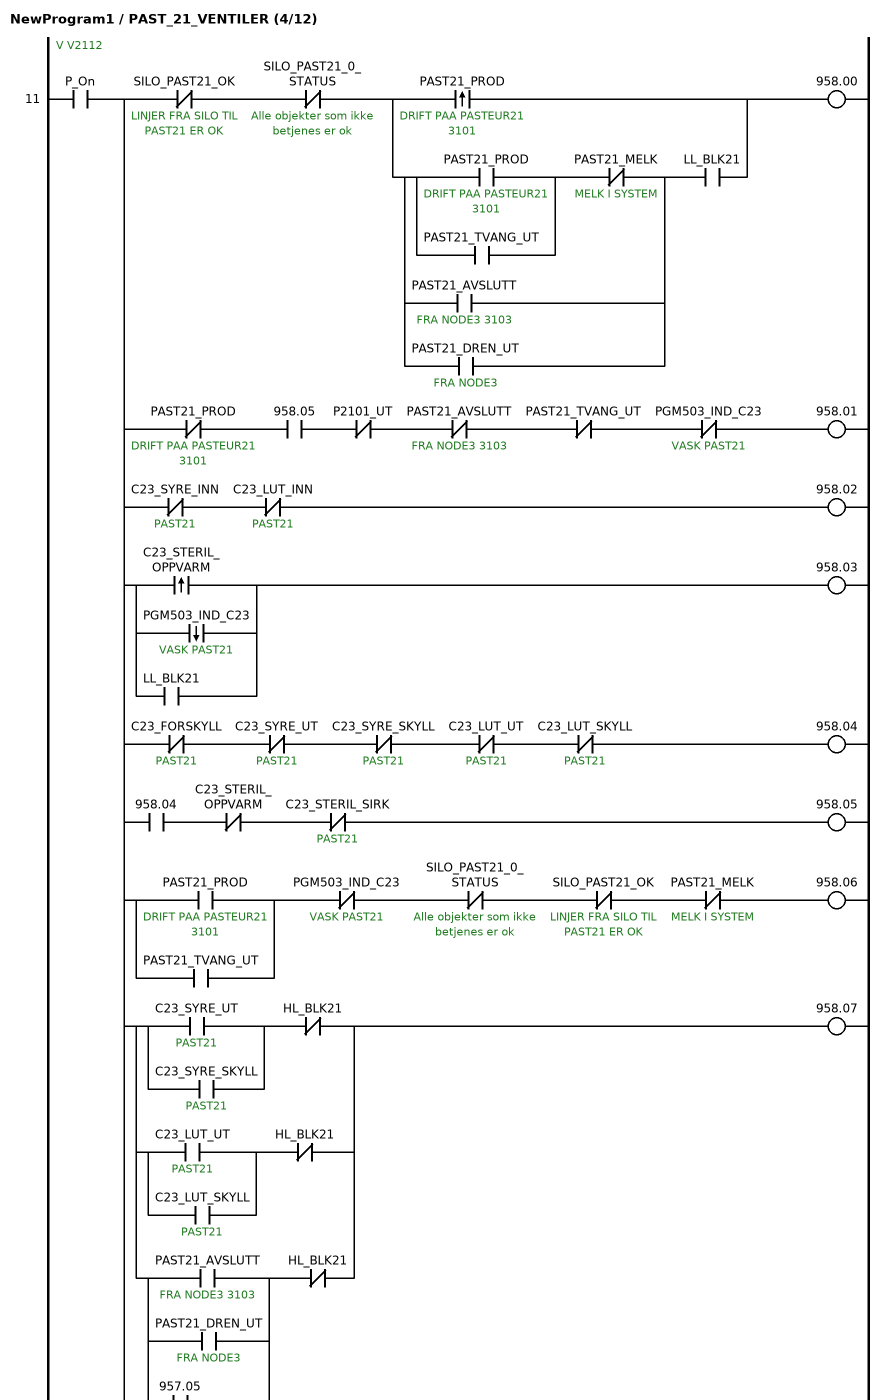
; [picture p1104: NewProgram1 / PAST_21_VENTILER, rungs 11-11]

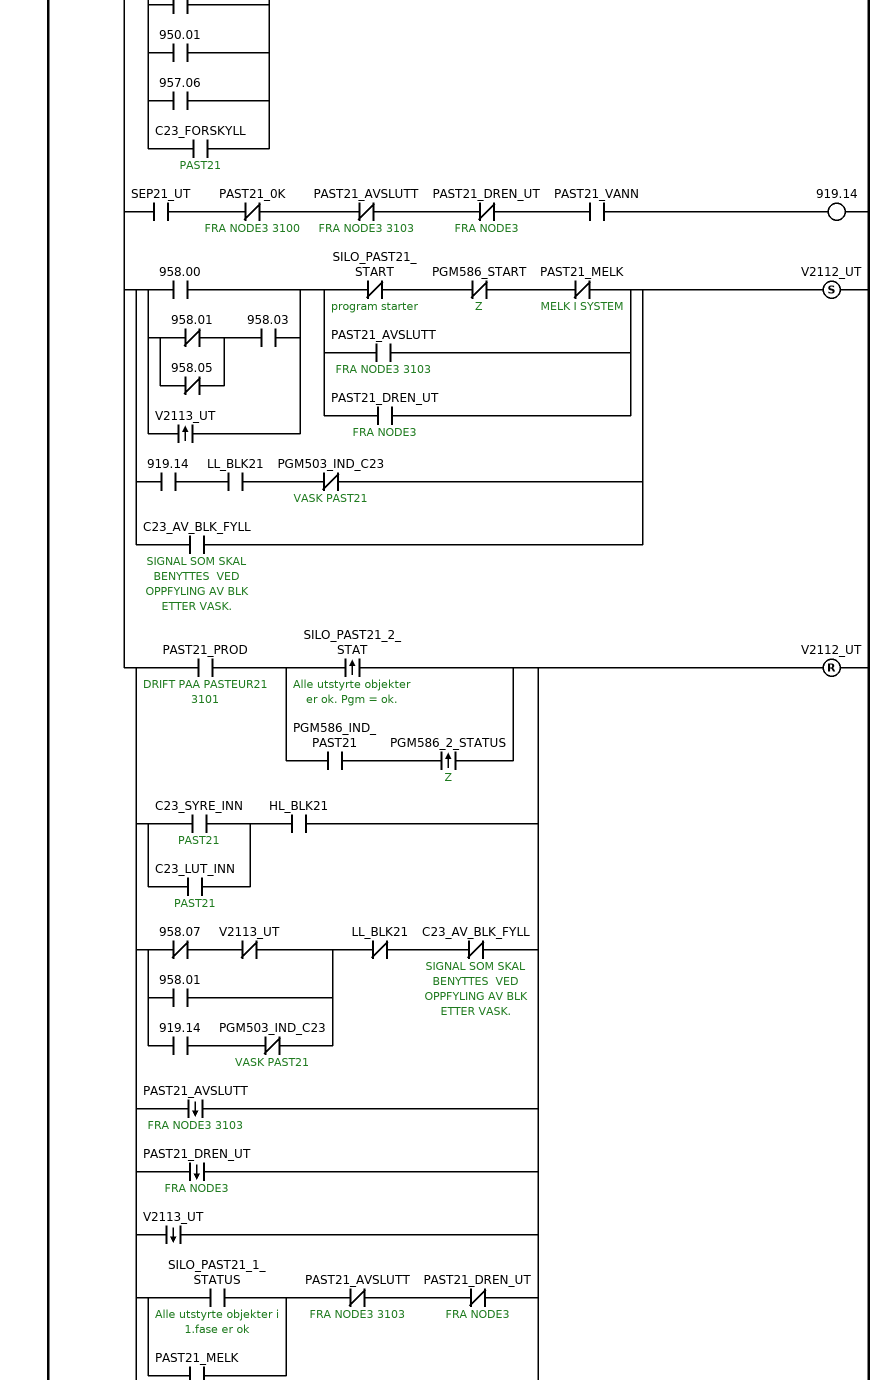

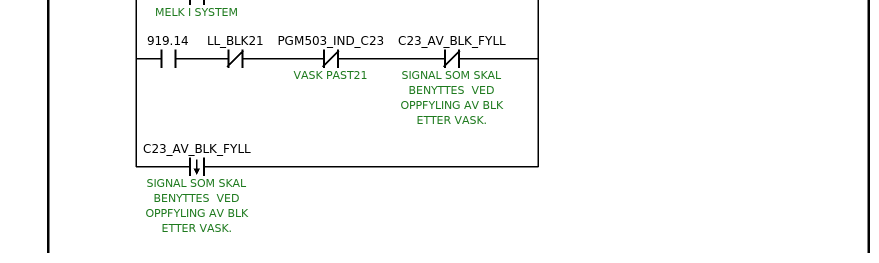
; rung 11: V V2112
LD P_On
OUT TR0
ANDNOT SILO_PAST21_OK  ; LINJER FRA SILO TIL  PAST21 ER OK
ANDNOT SILO_PAST21_0_STATUS  ; Alle objekter som ikke betjenes er ok
@LD PAST21_PROD  ; DRIFT PAA PASTEUR21 3101
LD PAST21_PROD  ; DRIFT PAA PASTEUR21 3101
OR PAST21_TVANG_UT
ANDNOT PAST21_MELK  ; MELK I SYSTEM
OR PAST21_AVSLUTT  ; FRA NODE3 3103
OR PAST21_DREN_UT  ; FRA NODE3
AND LL_BLK21
ORLD
ANDLD
OUT 958.00
LD TR0
ANDNOT PAST21_PROD  ; DRIFT PAA PASTEUR21 3101
AND 958.05
ANDNOT P2101_UT
ANDNOT PAST21_AVSLUTT  ; FRA NODE3 3103
ANDNOT PAST21_TVANG_UT
ANDNOT PGM503_IND_C23  ; VASK PAST21
OUT 958.01
LD TR0
ANDNOT C23_SYRE_INN  ; PAST21
ANDNOT C23_LUT_INN  ; PAST21
OUT 958.02
LD TR0
@LD C23_STERIL_OPPVARM
%OR PGM503_IND_C23  ; VASK PAST21
OR LL_BLK21
ANDLD
OUT 958.03
LD TR0
ANDNOT C23_FORSKYLL  ; PAST21
ANDNOT C23_SYRE_UT  ; PAST21
ANDNOT C23_SYRE_SKYLL  ; PAST21
ANDNOT C23_LUT_UT  ; PAST21
ANDNOT C23_LUT_SKYLL  ; PAST21
OUT 958.04
LD TR0
AND 958.04
ANDNOT C23_STERIL_OPPVARM
ANDNOT C23_STERIL_SIRK  ; PAST21
OUT 958.05
LD TR0
LD PAST21_PROD  ; DRIFT PAA PASTEUR21 3101
OR PAST21_TVANG_UT
ANDLD
ANDNOT PGM503_IND_C23  ; VASK PAST21
ANDNOT SILO_PAST21_0_STATUS  ; Alle objekter som ikke betjenes er ok
ANDNOT SILO_PAST21_OK  ; LINJER FRA SILO TIL  PAST21 ER OK
ANDNOT PAST21_MELK  ; MELK I SYSTEM
OUT 958.06
LD TR0
LD C23_SYRE_UT  ; PAST21
OR C23_SYRE_SKYLL  ; PAST21
ANDNOT HL_BLK21
LD C23_LUT_UT  ; PAST21
OR C23_LUT_SKYLL  ; PAST21
ANDNOT HL_BLK21
ORLD
LD PAST21_AVSLUTT  ; FRA NODE3 3103
OR PAST21_DREN_UT  ; FRA NODE3
OR 957.05
OR 950.01
OR 957.06
OR C23_FORSKYLL  ; PAST21
ANDNOT HL_BLK21
ORLD
ANDLD
OUT 958.07
LD TR0
AND SEP21_UT
ANDNOT PAST21_0K  ; FRA NODE3 3100
ANDNOT PAST21_AVSLUTT  ; FRA NODE3 3103
ANDNOT PAST21_DREN_UT  ; FRA NODE3
AND PAST21_VANN
OUT 919.14
LD TR0
LD 958.00
LDNOT 958.01
ORNOT 958.05
AND 958.03
ORLD
@OR V2113_UT
LDNOT SILO_PAST21_START  ; program starter
ANDNOT PGM586_START  ; Z
ANDNOT PAST21_MELK  ; MELK I SYSTEM
OR PAST21_AVSLUTT  ; FRA NODE3 3103
OR PAST21_DREN_UT  ; FRA NODE3
ANDLD
LD 919.14
AND LL_BLK21
ANDNOT PGM503_IND_C23  ; VASK PAST21
ORLD
OR C23_AV_BLK_FYLL  ; SIGNAL SOM SKAL BENYTTES  VED OPPFYLING AV BLK ETTER VASK.
ANDLD
SET V2112_UT
LD TR0
LD PAST21_PROD  ; DRIFT PAA PASTEUR21 3101
@LD SILO_PAST21_2_STAT  ; Alle utstyrte objekter er ok. Pgm = ok.
LD PGM586_IND_PAST21
@AND PGM586_2_STATUS  ; Z
ORLD
ANDLD
LD C23_SYRE_INN  ; PAST21
OR C23_LUT_INN  ; PAST21
AND HL_BLK21
ORLD
LDNOT 958.07
ANDNOT V2113_UT
OR 958.01
LD 919.14
ANDNOT PGM503_IND_C23  ; VASK PAST21
ORLD
ANDNOT LL_BLK21
ANDNOT C23_AV_BLK_FYLL  ; SIGNAL SOM SKAL BENYTTES  VED OPPFYLING AV BLK ETTER VASK.
ORLD
%OR PAST21_AVSLUTT  ; FRA NODE3 3103
%OR PAST21_DREN_UT  ; FRA NODE3
%OR V2113_UT
LD SILO_PAST21_1_STATUS  ; Alle utstyrte objekter i 1.fase er ok
OR PAST21_MELK  ; MELK I SYSTEM
ANDNOT PAST21_AVSLUTT  ; FRA NODE3 3103
ANDNOT PAST21_DREN_UT  ; FRA NODE3
ORLD
LD 919.14
ANDNOT LL_BLK21
ANDNOT PGM503_IND_C23  ; VASK PAST21
ANDNOT C23_AV_BLK_FYLL  ; SIGNAL SOM SKAL BENYTTES  VED OPPFYLING AV BLK ETTER VASK.
ORLD
%OR C23_AV_BLK_FYLL  ; SIGNAL SOM SKAL BENYTTES  VED OPPFYLING AV BLK ETTER VASK.
ANDLD
RSET V2112_UT

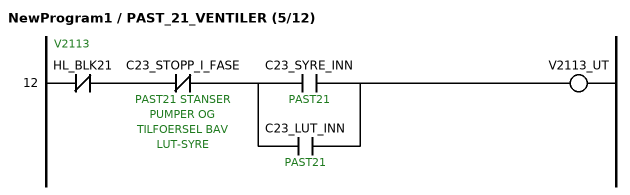
; rung 12: V2113
LDNOT HL_BLK21
ANDNOT C23_STOPP_I_FASE  ; PAST21 STANSER PUMPER OG TILFOERSEL BAV LUT-SYRE
LD C23_SYRE_INN  ; PAST21
OR C23_LUT_INN  ; PAST21
ANDLD
OUT V2113_UT

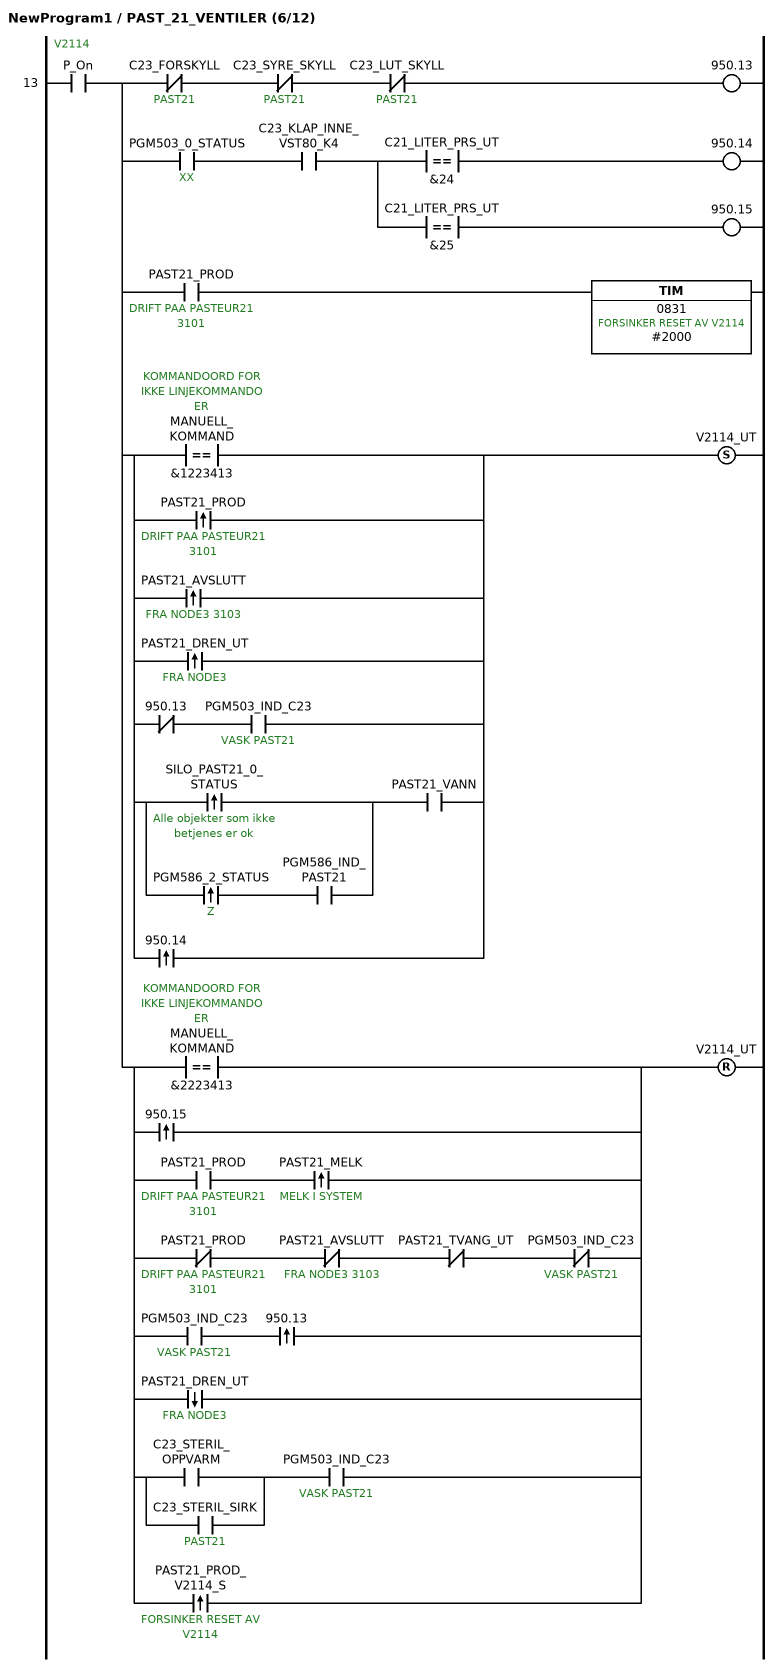
; rung 13: V2114
LD P_On
OUT TR0
ANDNOT C23_FORSKYLL  ; PAST21
ANDNOT C23_SYRE_SKYLL  ; PAST21
ANDNOT C23_LUT_SKYLL  ; PAST21
OUT 950.13
LD TR0
AND PGM503_0_STATUS  ; XX
AND C23_KLAP_INNE_VST80_K4
OUT TR1
AND=(300) C21_LITER_PRS_UT &24
OUT 950.14
LD TR1
AND=(300) C21_LITER_PRS_UT &25
OUT 950.15
LD TR0
AND PAST21_PROD  ; DRIFT PAA PASTEUR21 3101
TIM 0831 #2000  ; FORSINKER RESET AV V2114
LD TR0
LD=L(301) MANUELL_KOMMAND &1223413  ; KOMMANDOORD FOR IKKE LINJEKOMMANDOER
@OR PAST21_PROD  ; DRIFT PAA PASTEUR21 3101
@OR PAST21_AVSLUTT  ; FRA NODE3 3103
@OR PAST21_DREN_UT  ; FRA NODE3
LDNOT 950.13
AND PGM503_IND_C23  ; VASK PAST21
ORLD
@LD SILO_PAST21_0_STATUS  ; Alle objekter som ikke betjenes er ok
@LD PGM586_2_STATUS  ; Z
AND PGM586_IND_PAST21
ORLD
AND PAST21_VANN
ORLD
@OR 950.14
ANDLD
SET V2114_UT
LD TR0
LD=L(301) MANUELL_KOMMAND &2223413  ; KOMMANDOORD FOR IKKE LINJEKOMMANDOER
@OR 950.15
LD PAST21_PROD  ; DRIFT PAA PASTEUR21 3101
@AND PAST21_MELK  ; MELK I SYSTEM
ORLD
LDNOT PAST21_PROD  ; DRIFT PAA PASTEUR21 3101
ANDNOT PAST21_AVSLUTT  ; FRA NODE3 3103
ANDNOT PAST21_TVANG_UT
ANDNOT PGM503_IND_C23  ; VASK PAST21
ORLD
LD PGM503_IND_C23  ; VASK PAST21
@AND 950.13
ORLD
%OR PAST21_DREN_UT  ; FRA NODE3
LD C23_STERIL_OPPVARM
OR C23_STERIL_SIRK  ; PAST21
AND PGM503_IND_C23  ; VASK PAST21
ORLD
@OR PAST21_PROD_V2114_S  ; FORSINKER RESET AV V2114
ANDLD
RSET V2114_UT

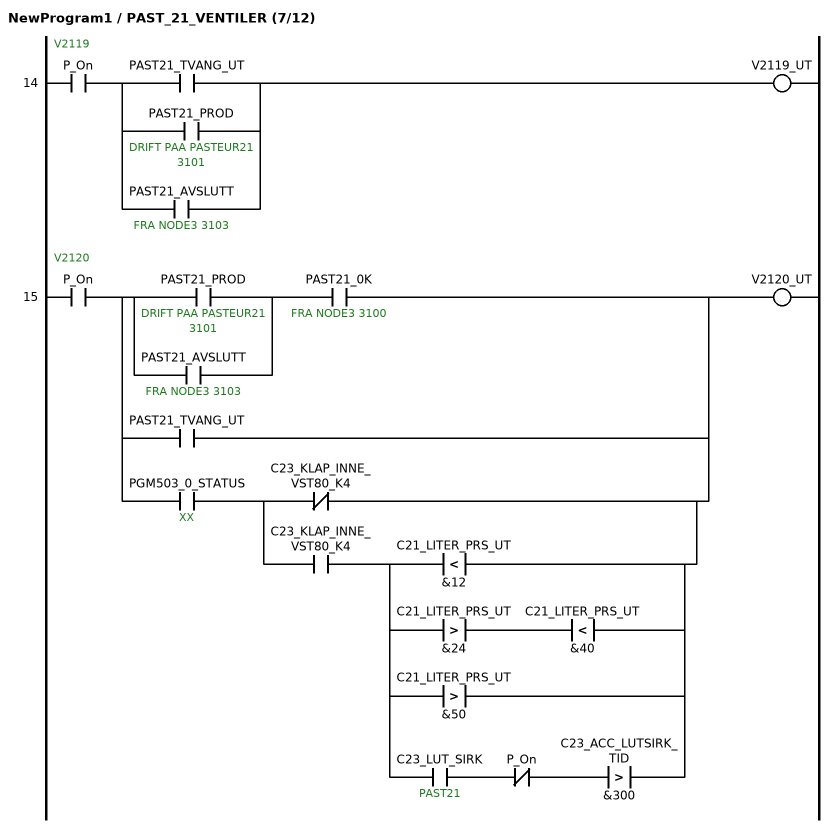
; rung 14: V2119
LD P_On
LD PAST21_TVANG_UT
OR PAST21_PROD  ; DRIFT PAA PASTEUR21 3101
OR PAST21_AVSLUTT  ; FRA NODE3 3103
ANDLD
OUT V2119_UT
; rung 15: V2120
LD P_On
LD PAST21_PROD  ; DRIFT PAA PASTEUR21 3101
OR PAST21_AVSLUTT  ; FRA NODE3 3103
AND PAST21_0K  ; FRA NODE3 3100
OR PAST21_TVANG_UT
LD PGM503_0_STATUS  ; XX
LDNOT C23_KLAP_INNE_VST80_K4
LD C23_KLAP_INNE_VST80_K4
LD<(310) C21_LITER_PRS_UT &12
LD>(320) C21_LITER_PRS_UT &24
AND<(310) C21_LITER_PRS_UT &40
ORLD
OR>(320) C21_LITER_PRS_UT &50
LD C23_LUT_SIRK  ; PAST21
ANDNOT P_On
AND>(320) C23_ACC_LUTSIRK_TID &300
ORLD
ANDLD
ORLD
ANDLD
ORLD
ANDLD
OUT V2120_UT

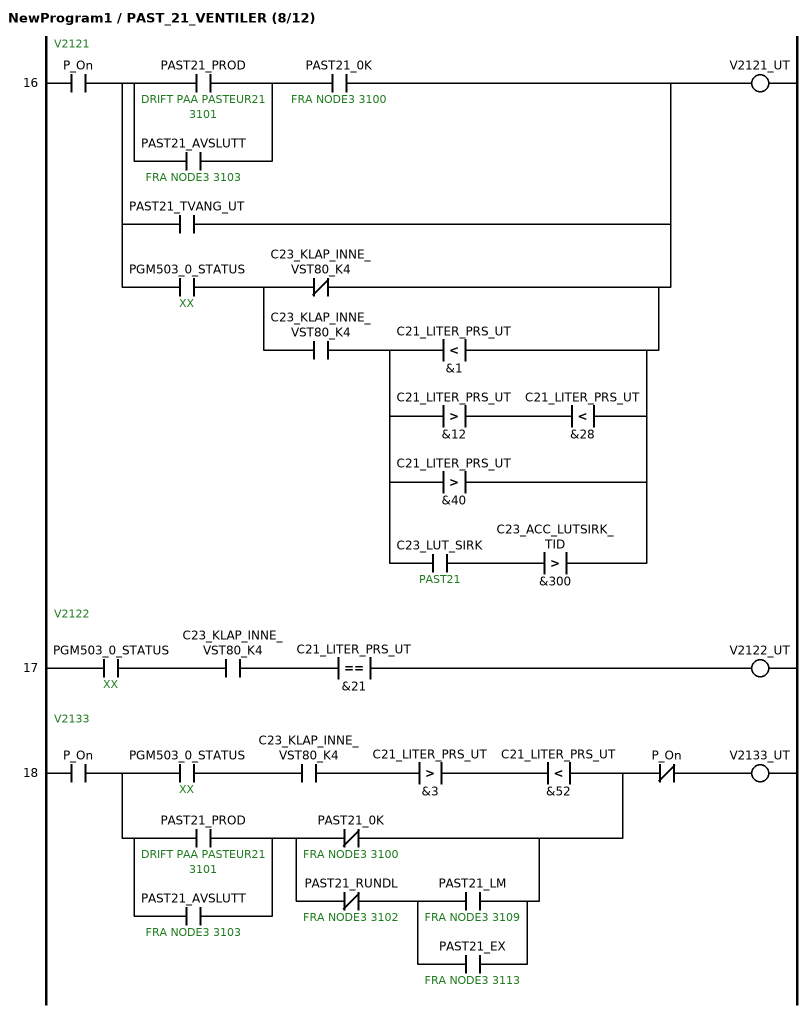
; rung 16: V2121
LD P_On
LD PAST21_PROD  ; DRIFT PAA PASTEUR21 3101
OR PAST21_AVSLUTT  ; FRA NODE3 3103
AND PAST21_0K  ; FRA NODE3 3100
OR PAST21_TVANG_UT
LD PGM503_0_STATUS  ; XX
LDNOT C23_KLAP_INNE_VST80_K4
LD C23_KLAP_INNE_VST80_K4
LD<(310) C21_LITER_PRS_UT &1
LD>(320) C21_LITER_PRS_UT &12
AND<(310) C21_LITER_PRS_UT &28
ORLD
OR>(320) C21_LITER_PRS_UT &40
LD C23_LUT_SIRK  ; PAST21
AND>(320) C23_ACC_LUTSIRK_TID &300
ORLD
ANDLD
ORLD
ANDLD
ORLD
ANDLD
OUT V2121_UT
; rung 17: V2122
LD PGM503_0_STATUS  ; XX
AND C23_KLAP_INNE_VST80_K4
AND=(300) C21_LITER_PRS_UT &21
OUT V2122_UT
; rung 18: V2133
LD P_On
LD PGM503_0_STATUS  ; XX
AND C23_KLAP_INNE_VST80_K4
AND>(320) C21_LITER_PRS_UT &3
AND<(310) C21_LITER_PRS_UT &52
LD PAST21_PROD  ; DRIFT PAA PASTEUR21 3101
OR PAST21_AVSLUTT  ; FRA NODE3 3103
LDNOT PAST21_0K  ; FRA NODE3 3100
LDNOT PAST21_RUNDL  ; FRA NODE3 3102
LD PAST21_LM  ; FRA NODE3 3109
OR PAST21_EX  ; FRA NODE3 3113
ANDLD
ORLD
ANDLD
ORLD
ANDLD
ANDNOT P_On
OUT V2133_UT

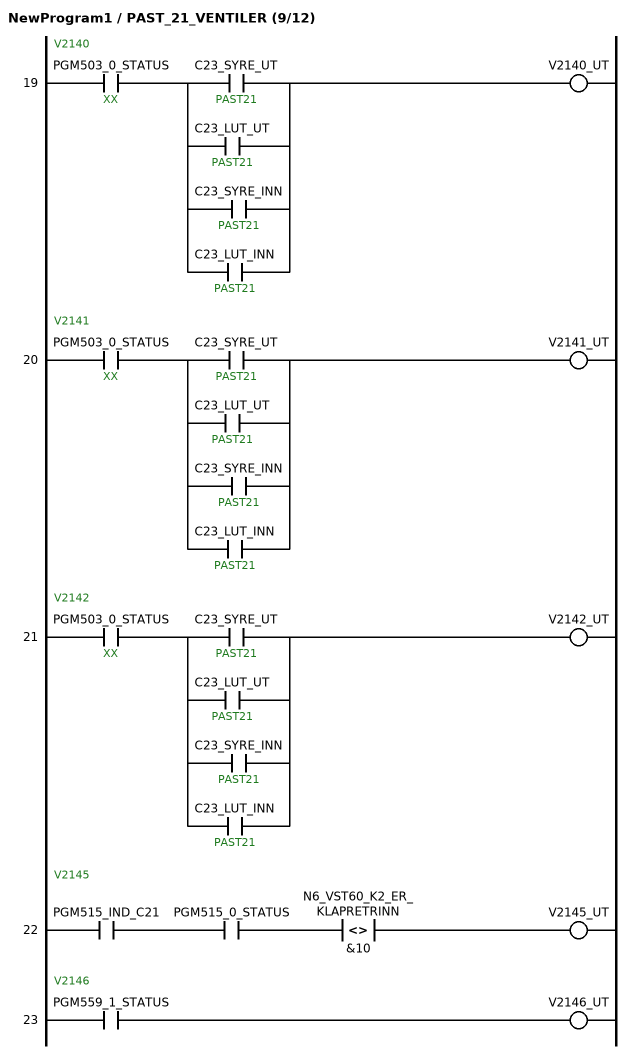
; rung 19: V2140
LD PGM503_0_STATUS  ; XX
LD C23_SYRE_UT  ; PAST21
OR C23_LUT_UT  ; PAST21
OR C23_SYRE_INN  ; PAST21
OR C23_LUT_INN  ; PAST21
ANDLD
OUT V2140_UT
; rung 20: V2141
LD PGM503_0_STATUS  ; XX
LD C23_SYRE_UT  ; PAST21
OR C23_LUT_UT  ; PAST21
OR C23_SYRE_INN  ; PAST21
OR C23_LUT_INN  ; PAST21
ANDLD
OUT V2141_UT
; rung 21: V2142
LD PGM503_0_STATUS  ; XX
LD C23_SYRE_UT  ; PAST21
OR C23_LUT_UT  ; PAST21
OR C23_SYRE_INN  ; PAST21
OR C23_LUT_INN  ; PAST21
ANDLD
OUT V2142_UT
; rung 22: V2145
LD PGM515_IND_C21
AND PGM515_0_STATUS
AND<>(305) N6_VST60_K2_ER_KLAPRETRINN &10
OUT V2145_UT
; rung 23: V2146
LD PGM559_1_STATUS
OUT V2146_UT

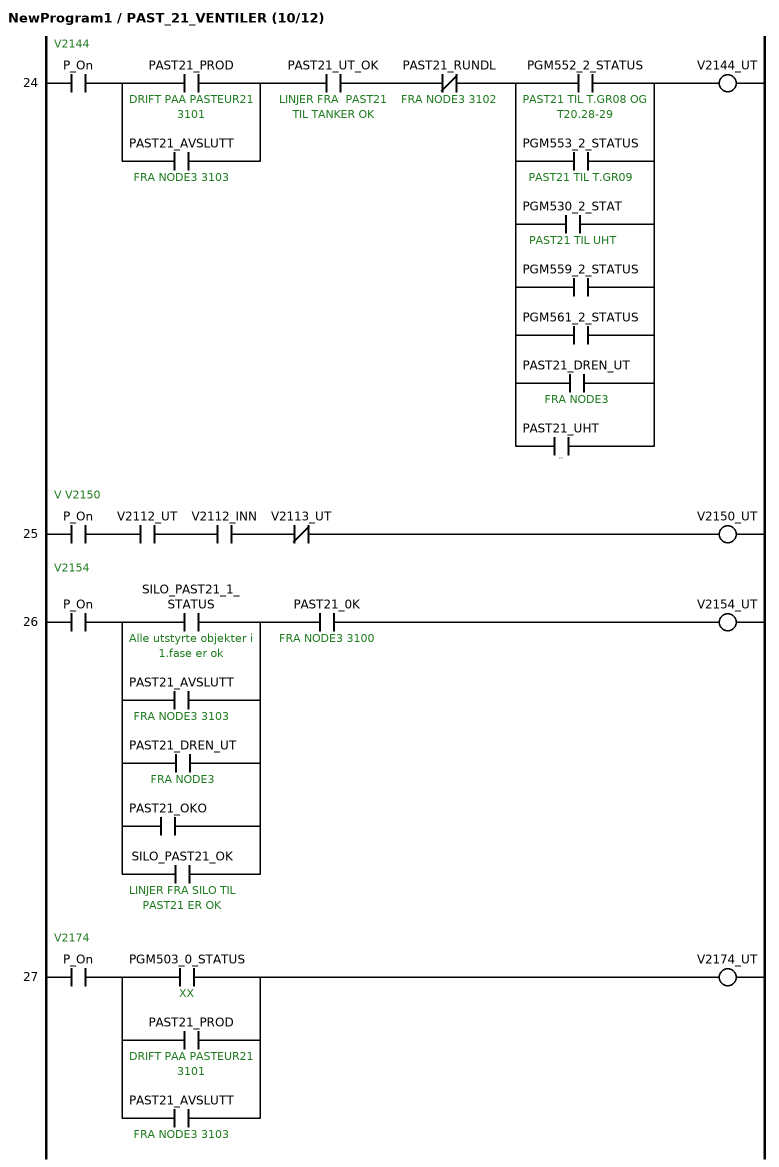
; rung 24: V2144
LD P_On
LD PAST21_PROD  ; DRIFT PAA PASTEUR21 3101
OR PAST21_AVSLUTT  ; FRA NODE3 3103
ANDLD
AND PAST21_UT_OK  ; LINJER FRA  PAST21 TIL TANKER OK
ANDNOT PAST21_RUNDL  ; FRA NODE3 3102
LD PGM552_2_STATUS  ; PAST21 TIL T.GR08 OG T20.28-29
OR PGM553_2_STATUS  ; PAST21 TIL T.GR09
OR PGM530_2_STAT  ; PAST21 TIL UHT
OR PGM559_2_STATUS
OR PGM561_2_STATUS
OR PAST21_DREN_UT  ; FRA NODE3
OR PAST21_UHT  ; ¨
ANDLD
OUT V2144_UT
; rung 25: V V2150
LD P_On
AND V2112_UT
AND V2112_INN
ANDNOT V2113_UT
OUT V2150_UT
; rung 26: V2154
LD P_On
LD SILO_PAST21_1_STATUS  ; Alle utstyrte objekter i 1.fase er ok
OR PAST21_AVSLUTT  ; FRA NODE3 3103
OR PAST21_DREN_UT  ; FRA NODE3
OR PAST21_OKO
OR SILO_PAST21_OK  ; LINJER FRA SILO TIL  PAST21 ER OK
ANDLD
AND PAST21_0K  ; FRA NODE3 3100
OUT V2154_UT
; rung 27: V2174
LD P_On
LD PGM503_0_STATUS  ; XX
OR PAST21_PROD  ; DRIFT PAA PASTEUR21 3101
OR PAST21_AVSLUTT  ; FRA NODE3 3103
ANDLD
OUT V2174_UT

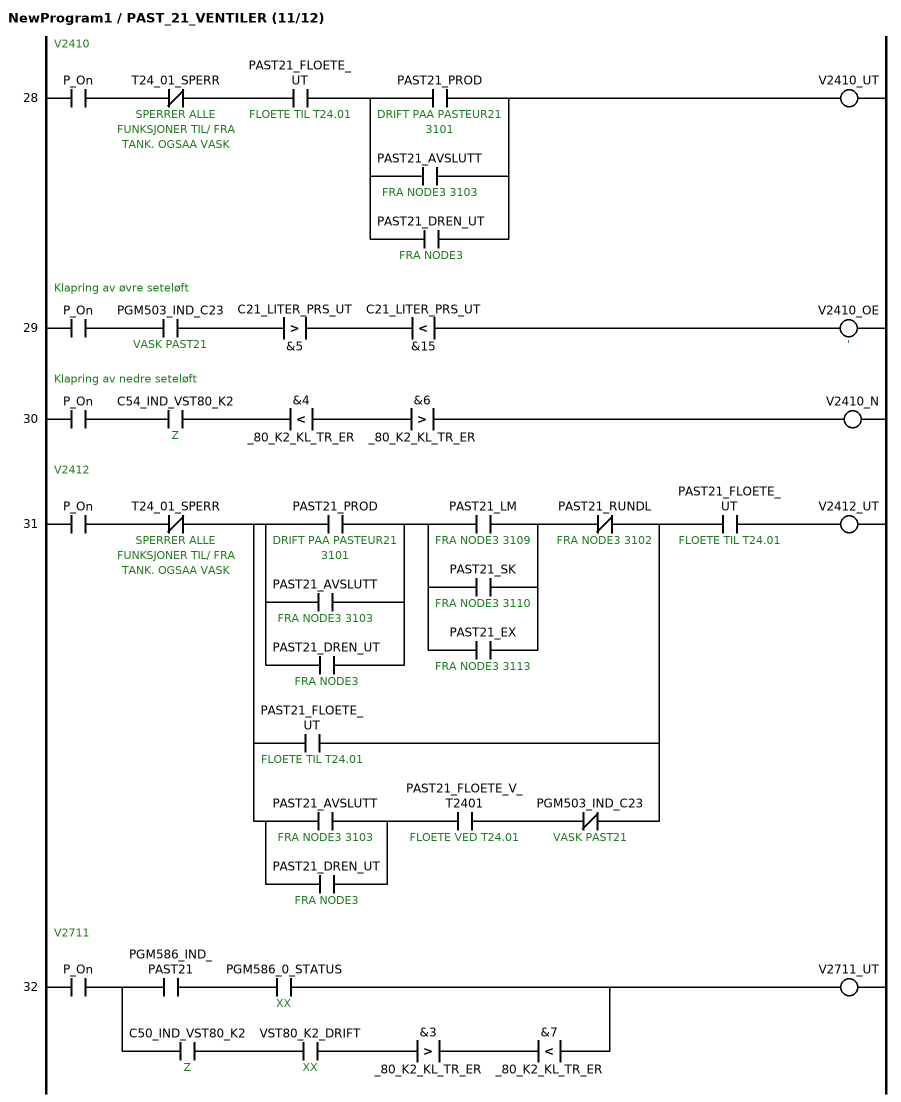
; rung 28: V2410
LD P_On
ANDNOT T24_01_SPERR  ; SPERRER ALLE FUNKSJONER TIL/ FRA TANK. OGSAA VASK
AND PAST21_FLOETE_UT  ; FLOETE TIL T24.01
LD PAST21_PROD  ; DRIFT PAA PASTEUR21 3101
OR PAST21_AVSLUTT  ; FRA NODE3 3103
OR PAST21_DREN_UT  ; FRA NODE3
ANDLD
OUT V2410_UT
; rung 29: Klapring av øvre seteløft
LD P_On
AND PGM503_IND_C23  ; VASK PAST21
AND>(320) C21_LITER_PRS_UT &5
AND<(310) C21_LITER_PRS_UT &15
OUT V2410_OE  ; '
; rung 30: Klapring av nedre seteløft
LD P_On
AND C54_IND_VST80_K2  ; Z
AND<(310) &4 _80_K2_KL_TR_ER
AND>(320) &6 _80_K2_KL_TR_ER
OUT V2410_N
; rung 31: V2412
LD P_On
ANDNOT T24_01_SPERR  ; SPERRER ALLE FUNKSJONER TIL/ FRA TANK. OGSAA VASK
LD PAST21_PROD  ; DRIFT PAA PASTEUR21 3101
OR PAST21_AVSLUTT  ; FRA NODE3 3103
OR PAST21_DREN_UT  ; FRA NODE3
LD PAST21_LM  ; FRA NODE3 3109
OR PAST21_SK  ; FRA NODE3 3110
OR PAST21_EX  ; FRA NODE3 3113
ANDLD
ANDNOT PAST21_RUNDL  ; FRA NODE3 3102
OR PAST21_FLOETE_UT  ; FLOETE TIL T24.01
LD PAST21_AVSLUTT  ; FRA NODE3 3103
OR PAST21_DREN_UT  ; FRA NODE3
AND PAST21_FLOETE_V_T2401  ; FLOETE VED T24.01
ANDNOT PGM503_IND_C23  ; VASK PAST21
ORLD
ANDLD
AND PAST21_FLOETE_UT  ; FLOETE TIL T24.01
OUT V2412_UT
; rung 32: V2711
LD P_On
LD PGM586_IND_PAST21
AND PGM586_0_STATUS  ; XX
LD C50_IND_VST80_K2  ; Z
AND VST80_K2_DRIFT  ; XX
AND>(320) &3 _80_K2_KL_TR_ER
AND<(310) &7 _80_K2_KL_TR_ER
ORLD
ANDLD
OUT V2711_UT

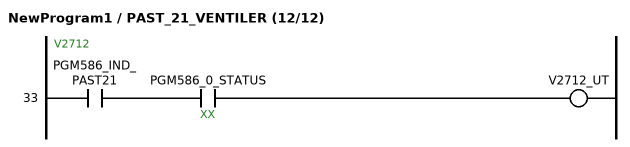
; rung 33: V2712
LD PGM586_IND_PAST21
AND PGM586_0_STATUS  ; XX
OUT V2712_UT

### Section PAST_21_SKRIVER

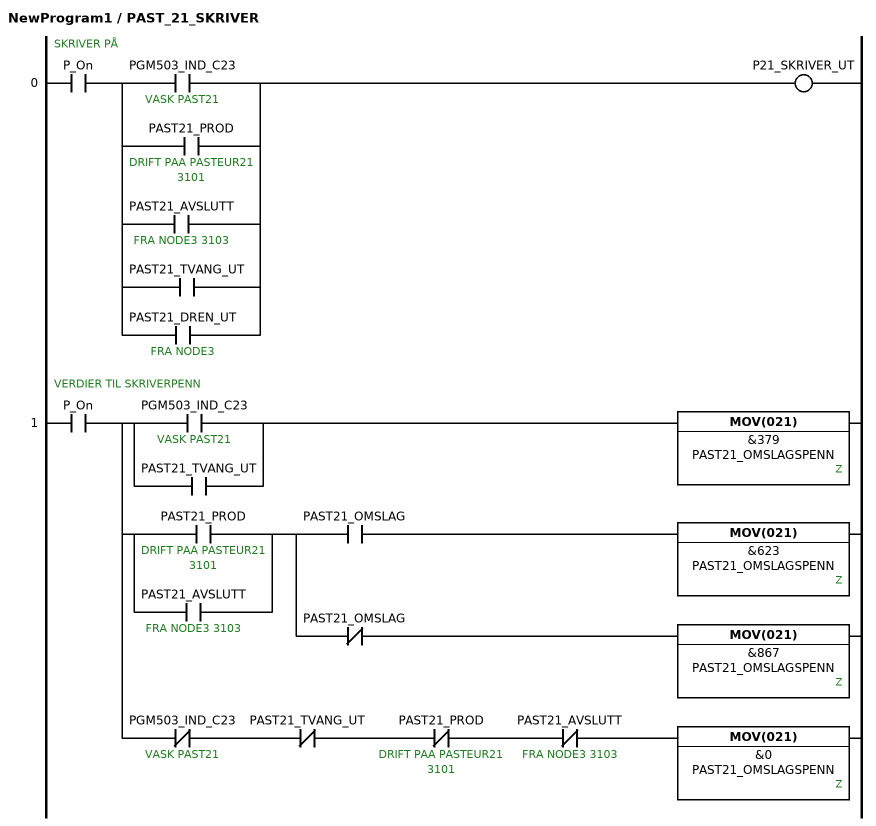
; rung 0: SKRIVER PÅ
LD P_On
LD PGM503_IND_C23  ; VASK PAST21
OR PAST21_PROD  ; DRIFT PAA PASTEUR21 3101
OR PAST21_AVSLUTT  ; FRA NODE3 3103
OR PAST21_TVANG_UT
OR PAST21_DREN_UT  ; FRA NODE3
ANDLD
OUT P21_SKRIVER_UT
; rung 1: VERDIER TIL SKRIVERPENN
LD P_On
OUT TR0
LD PGM503_IND_C23  ; VASK PAST21
OR PAST21_TVANG_UT
ANDLD
MOV(021) &379 PAST21_OMSLAGSPENN  ; Z
LD TR0
LD PAST21_PROD  ; DRIFT PAA PASTEUR21 3101
OR PAST21_AVSLUTT  ; FRA NODE3 3103
ANDLD
OUT TR1
AND PAST21_OMSLAG
MOV(021) &623 PAST21_OMSLAGSPENN  ; Z
LD TR1
ANDNOT PAST21_OMSLAG
MOV(021) &867 PAST21_OMSLAGSPENN  ; Z
LD TR0
ANDNOT PGM503_IND_C23  ; VASK PAST21
ANDNOT PAST21_TVANG_UT
ANDNOT PAST21_PROD  ; DRIFT PAA PASTEUR21 3101
ANDNOT PAST21_AVSLUTT  ; FRA NODE3 3103
MOV(021) &0 PAST21_OMSLAGSPENN  ; Z

### Section PAST_21_TELLERFUNKSJONER

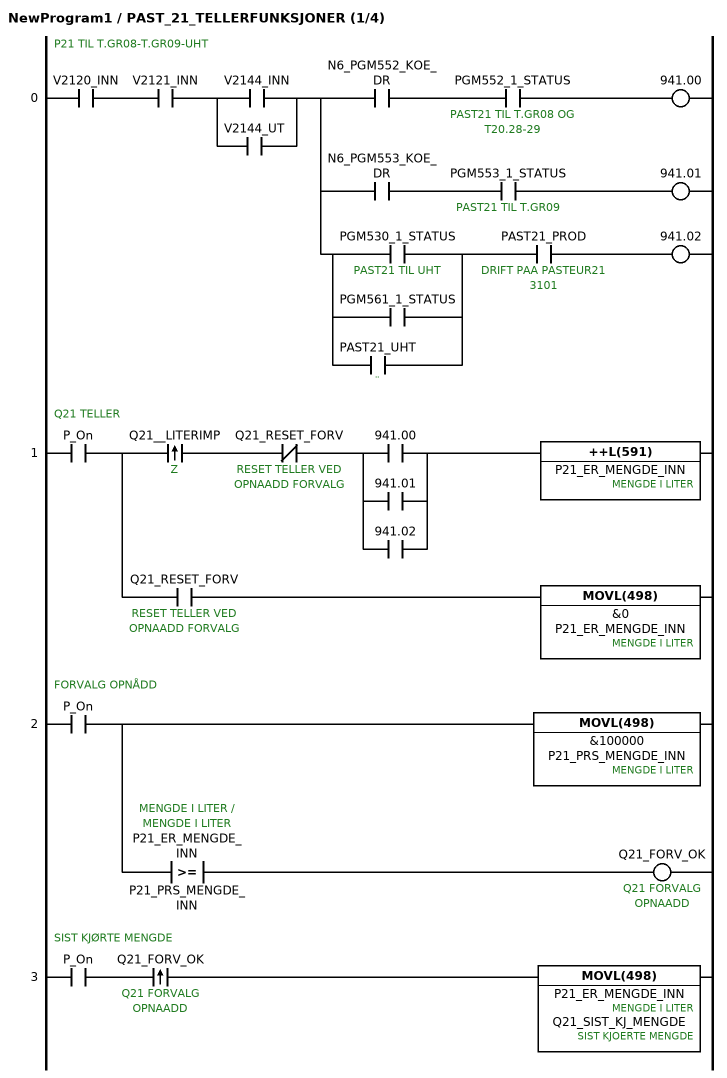
; rung 0: P21 TIL T.GR08-T.GR09-UHT
LD V2120_INN
AND V2121_INN
LD V2144_INN
OR V2144_UT
ANDLD
OUT TR0
AND N6_PGM552_KOE_DR
AND PGM552_1_STATUS  ; PAST21 TIL T.GR08 OG T20.28-29
OUT 941.00
LD TR0
AND N6_PGM553_KOE_DR
AND PGM553_1_STATUS  ; PAST21 TIL T.GR09
OUT 941.01
LD TR0
LD PGM530_1_STATUS  ; PAST21 TIL UHT
OR PGM561_1_STATUS
OR PAST21_UHT  ; ¨
ANDLD
AND PAST21_PROD  ; DRIFT PAA PASTEUR21 3101
OUT 941.02
; rung 1: Q21 TELLER
LD P_On
OUT TR0
@AND Q21__LITERIMP  ; Z
ANDNOT Q21_RESET_FORV  ; RESET TELLER VED OPNAADD FORVALG
LD 941.00
OR 941.01
OR 941.02
ANDLD
++L(591) P21_ER_MENGDE_INN  ; MENGDE I LITER
LD TR0
AND Q21_RESET_FORV  ; RESET TELLER VED OPNAADD FORVALG
MOVL(498) &0 P21_ER_MENGDE_INN  ; MENGDE I LITER
; rung 2: FORVALG OPNÅDD
LD P_On
MOVL(498) &100000 P21_PRS_MENGDE_INN  ; MENGDE I LITER
AND>=L(326) P21_ER_MENGDE_INN P21_PRS_MENGDE_INN  ; MENGDE I LITER
OUT Q21_FORV_OK  ; Q21 FORVALG OPNAADD
; rung 3: SIST KJØRTE MENGDE
LD P_On
@AND Q21_FORV_OK  ; Q21 FORVALG OPNAADD
MOVL(498) P21_ER_MENGDE_INN Q21_SIST_KJ_MENGDE  ; MENGDE I LITER, SIST KJOERTE MENGDE

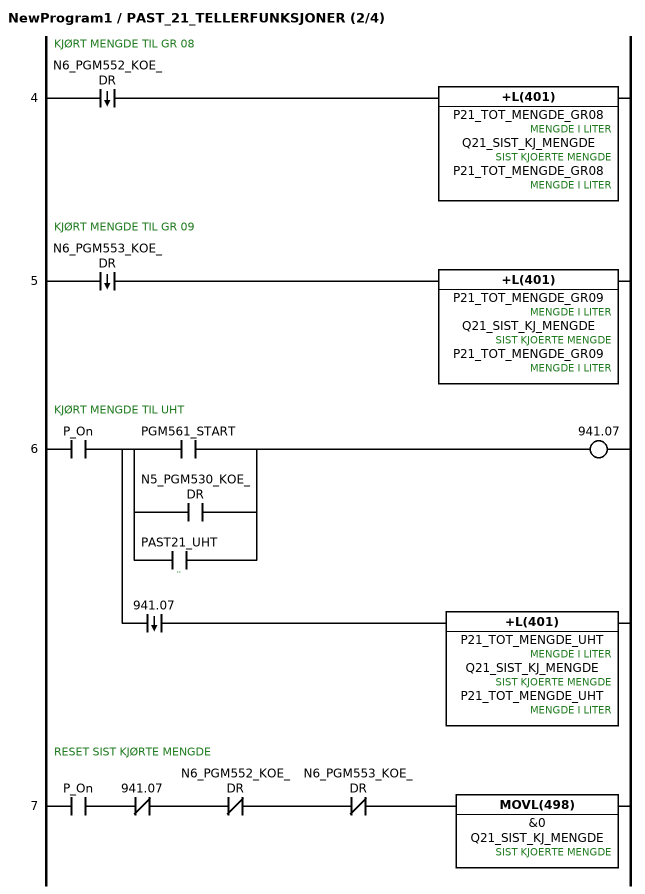
; rung 4: KJØRT MENGDE TIL GR 08
%LD N6_PGM552_KOE_DR
+L(401) P21_TOT_MENGDE_GR08 Q21_SIST_KJ_MENGDE P21_TOT_MENGDE_GR08  ; MENGDE I LITER, SIST KJOERTE MENGDE
; rung 5: KJØRT MENGDE TIL GR 09
%LD N6_PGM553_KOE_DR
+L(401) P21_TOT_MENGDE_GR09 Q21_SIST_KJ_MENGDE P21_TOT_MENGDE_GR09  ; MENGDE I LITER, SIST KJOERTE MENGDE
; rung 6: KJØRT MENGDE TIL UHT
LD P_On
OUT TR0
LD PGM561_START
OR N5_PGM530_KOE_DR
OR PAST21_UHT  ; ¨
ANDLD
OUT 941.07
LD TR0
%AND 941.07
+L(401) P21_TOT_MENGDE_UHT Q21_SIST_KJ_MENGDE P21_TOT_MENGDE_UHT  ; MENGDE I LITER, SIST KJOERTE MENGDE
; rung 7: RESET SIST KJØRTE MENGDE
LD P_On
ANDNOT 941.07
ANDNOT N6_PGM552_KOE_DR
ANDNOT N6_PGM553_KOE_DR
MOVL(498) &0 Q21_SIST_KJ_MENGDE  ; SIST KJOERTE MENGDE

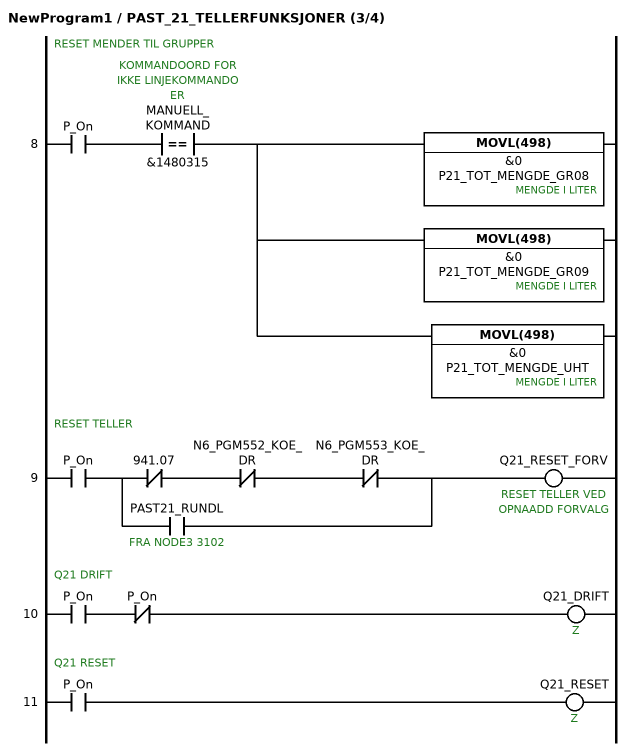
; rung 8: RESET MENDER TIL GRUPPER
LD P_On
AND=L(301) MANUELL_KOMMAND &1480315  ; KOMMANDOORD FOR IKKE LINJEKOMMANDOER
MOVL(498) &0 P21_TOT_MENGDE_GR08  ; MENGDE I LITER
MOVL(498) &0 P21_TOT_MENGDE_GR09  ; MENGDE I LITER
MOVL(498) &0 P21_TOT_MENGDE_UHT  ; MENGDE I LITER
; rung 9: RESET TELLER
LD P_On
LDNOT 941.07
ANDNOT N6_PGM552_KOE_DR
ANDNOT N6_PGM553_KOE_DR
OR PAST21_RUNDL  ; FRA NODE3 3102
ANDLD
OUT Q21_RESET_FORV  ; RESET TELLER VED OPNAADD FORVALG
; rung 10: Q21 DRIFT
LD P_On
ANDNOT P_On
OUT Q21_DRIFT  ; Z
; rung 11: Q21 RESET
LD P_On
OUT Q21_RESET  ; Z

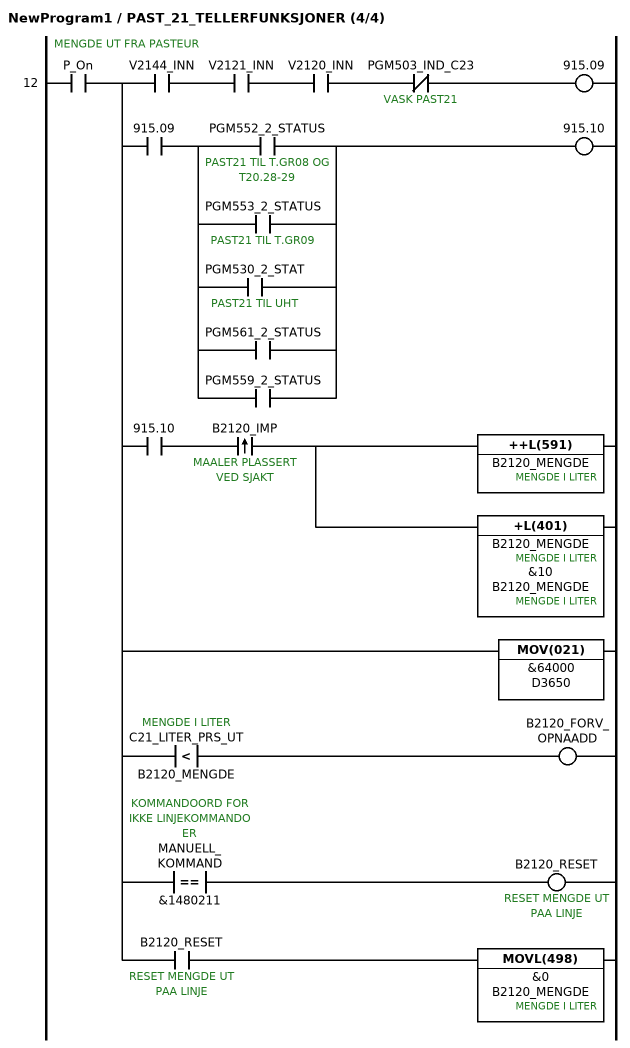
; rung 12: MENGDE UT FRA PASTEUR
LD P_On
OUT TR0
AND V2144_INN
AND V2121_INN
AND V2120_INN
ANDNOT PGM503_IND_C23  ; VASK PAST21
OUT 915.09
LD TR0
AND 915.09
LD PGM552_2_STATUS  ; PAST21 TIL T.GR08 OG T20.28-29
OR PGM553_2_STATUS  ; PAST21 TIL T.GR09
OR PGM530_2_STAT  ; PAST21 TIL UHT
OR PGM561_2_STATUS
OR PGM559_2_STATUS
ANDLD
OUT 915.10
LD TR0
AND 915.10
@AND B2120_IMP  ; MAALER PLASSERT VED SJAKT
++L(591) B2120_MENGDE  ; MENGDE I LITER
+L(401) B2120_MENGDE &10 B2120_MENGDE  ; MENGDE I LITER
LD TR0
MOV(021) &64000 D3650
AND<L(311) C21_LITER_PRS_UT B2120_MENGDE  ; MENGDE I LITER
OUT B2120_FORV_OPNAADD
LD TR0
AND=L(301) MANUELL_KOMMAND &1480211  ; KOMMANDOORD FOR IKKE LINJEKOMMANDOER
OUT B2120_RESET  ; RESET MENGDE UT PAA LINJE
LD TR0
AND B2120_RESET  ; RESET MENGDE UT PAA LINJE
MOVL(498) &0 B2120_MENGDE  ; MENGDE I LITER

### Section P21_MELK_IRØR_TIL_TGR

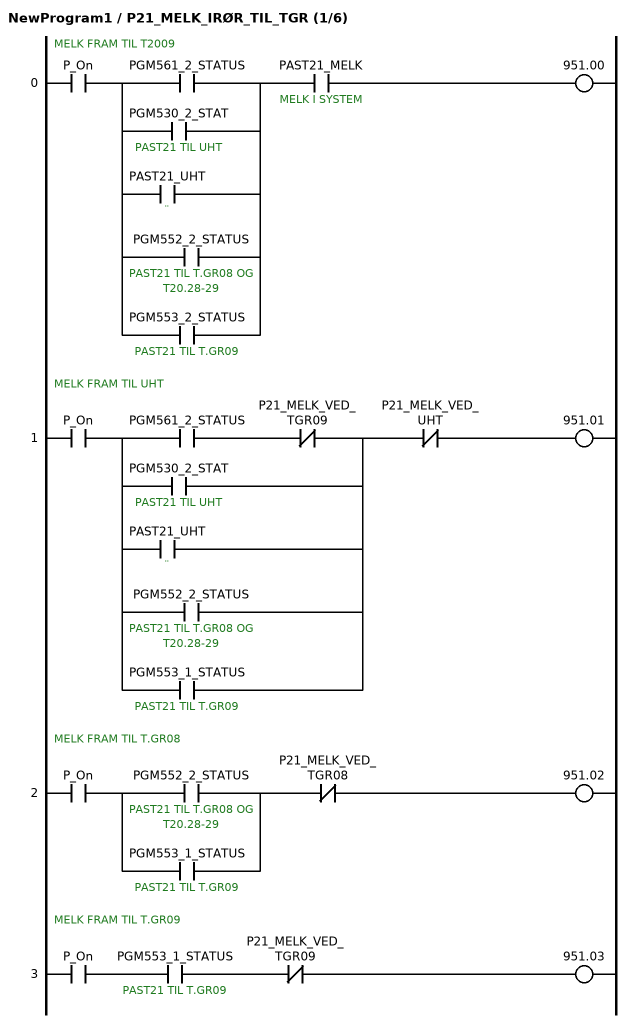
; rung 0: MELK FRAM TIL T2009
LD P_On
LD PGM561_2_STATUS
OR PGM530_2_STAT  ; PAST21 TIL UHT
OR PAST21_UHT  ; ¨
OR PGM552_2_STATUS  ; PAST21 TIL T.GR08 OG T20.28-29
OR PGM553_2_STATUS  ; PAST21 TIL T.GR09
ANDLD
AND PAST21_MELK  ; MELK I SYSTEM
OUT 951.00
; rung 1: MELK FRAM TIL UHT
LD P_On
LD PGM561_2_STATUS
ANDNOT P21_MELK_VED_TGR09
OR PGM530_2_STAT  ; PAST21 TIL UHT
OR PAST21_UHT  ; ¨
OR PGM552_2_STATUS  ; PAST21 TIL T.GR08 OG T20.28-29
OR PGM553_1_STATUS  ; PAST21 TIL T.GR09
ANDLD
ANDNOT P21_MELK_VED_UHT
OUT 951.01
; rung 2: MELK FRAM TIL T.GR08
LD P_On
LD PGM552_2_STATUS  ; PAST21 TIL T.GR08 OG T20.28-29
OR PGM553_1_STATUS  ; PAST21 TIL T.GR09
ANDLD
ANDNOT P21_MELK_VED_TGR08
OUT 951.02
; rung 3: MELK FRAM TIL T.GR09
LD P_On
AND PGM553_1_STATUS  ; PAST21 TIL T.GR09
ANDNOT P21_MELK_VED_TGR09
OUT 951.03

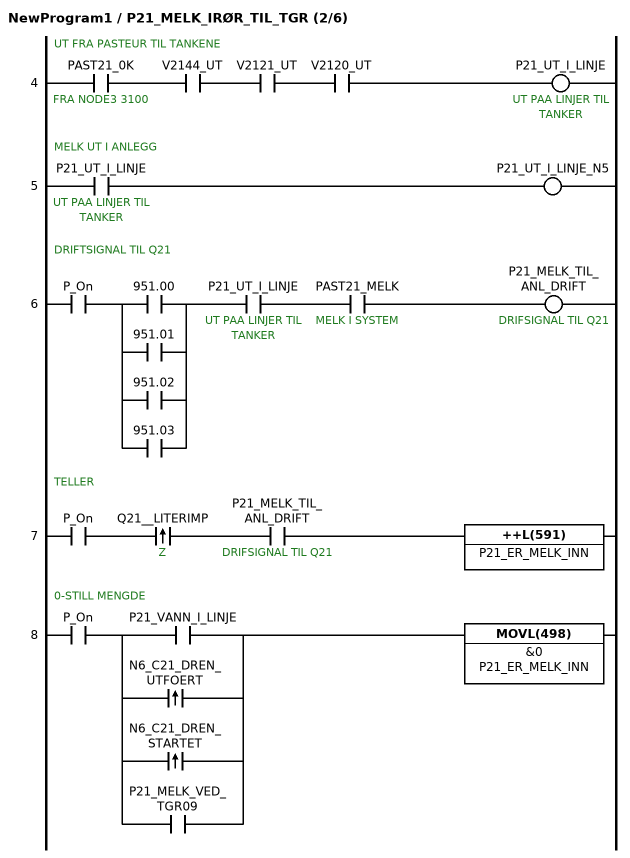
; rung 4: UT FRA PASTEUR TIL TANKENE
LD PAST21_0K  ; FRA NODE3 3100
AND V2144_UT
AND V2121_UT
AND V2120_UT
OUT P21_UT_I_LINJE  ; UT PAA LINJER TIL TANKER
; rung 5: MELK UT I ANLEGG
LD P21_UT_I_LINJE  ; UT PAA LINJER TIL TANKER
OUT P21_UT_I_LINJE_N5
; rung 6: DRIFTSIGNAL TIL Q21
LD P_On
LD 951.00
OR 951.01
OR 951.02
OR 951.03
ANDLD
AND P21_UT_I_LINJE  ; UT PAA LINJER TIL TANKER
AND PAST21_MELK  ; MELK I SYSTEM
OUT P21_MELK_TIL_ANL_DRIFT  ; DRIFSIGNAL TIL Q21
; rung 7: TELLER
LD P_On
@AND Q21__LITERIMP  ; Z
AND P21_MELK_TIL_ANL_DRIFT  ; DRIFSIGNAL TIL Q21
++L(591) P21_ER_MELK_INN
; rung 8: 0-STILL MENGDE
LD P_On
LD P21_VANN_I_LINJE
@OR N6_C21_DREN_UTFOERT
@OR N6_C21_DREN_STARTET
OR P21_MELK_VED_TGR09
ANDLD
MOVL(498) &0 P21_ER_MELK_INN

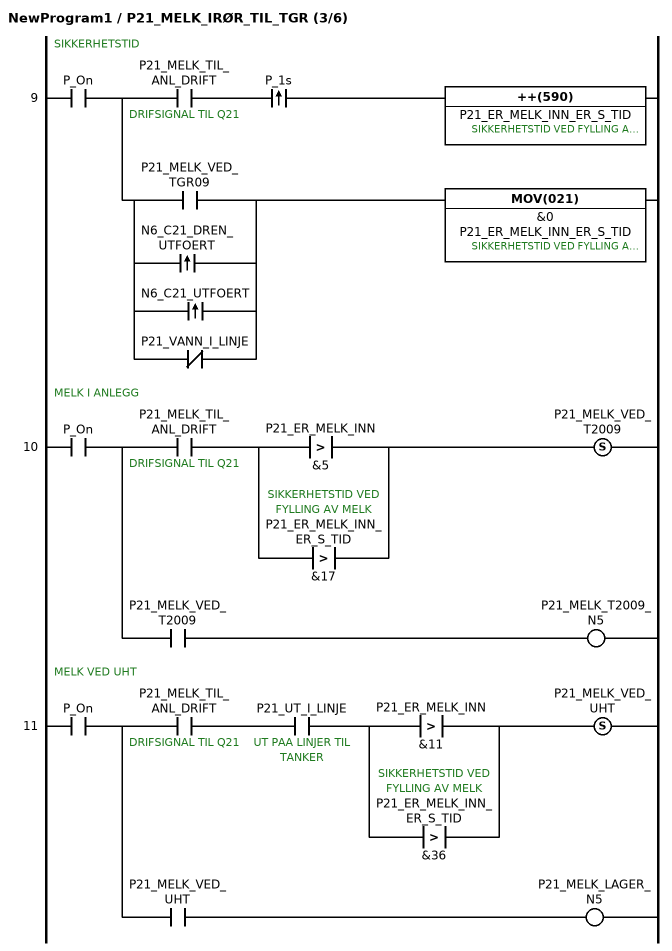
; rung 9: SIKKERHETSTID
LD P_On
OUT TR0
AND P21_MELK_TIL_ANL_DRIFT  ; DRIFSIGNAL TIL Q21
@AND P_1s
++(590) P21_ER_MELK_INN_ER_S_TID  ; SIKKERHETSTID VED FYLLING AV MELK
LD TR0
LD P21_MELK_VED_TGR09
@OR N6_C21_DREN_UTFOERT
@OR N6_C21_UTFOERT
ORNOT P21_VANN_I_LINJE
ANDLD
MOV(021) &0 P21_ER_MELK_INN_ER_S_TID  ; SIKKERHETSTID VED FYLLING AV MELK
; rung 10: MELK I ANLEGG
LD P_On
OUT TR0
AND P21_MELK_TIL_ANL_DRIFT  ; DRIFSIGNAL TIL Q21
LD>L(321) P21_ER_MELK_INN &5
OR>(320) P21_ER_MELK_INN_ER_S_TID &17  ; SIKKERHETSTID VED FYLLING AV MELK
ANDLD
SET P21_MELK_VED_T2009
LD TR0
AND P21_MELK_VED_T2009
OUT P21_MELK_T2009_N5
; rung 11: MELK VED UHT
LD P_On
OUT TR0
AND P21_MELK_TIL_ANL_DRIFT  ; DRIFSIGNAL TIL Q21
AND P21_UT_I_LINJE  ; UT PAA LINJER TIL TANKER
LD>L(321) P21_ER_MELK_INN &11
OR>(320) P21_ER_MELK_INN_ER_S_TID &36  ; SIKKERHETSTID VED FYLLING AV MELK
ANDLD
SET P21_MELK_VED_UHT
LD TR0
AND P21_MELK_VED_UHT
OUT P21_MELK_LAGER_N5

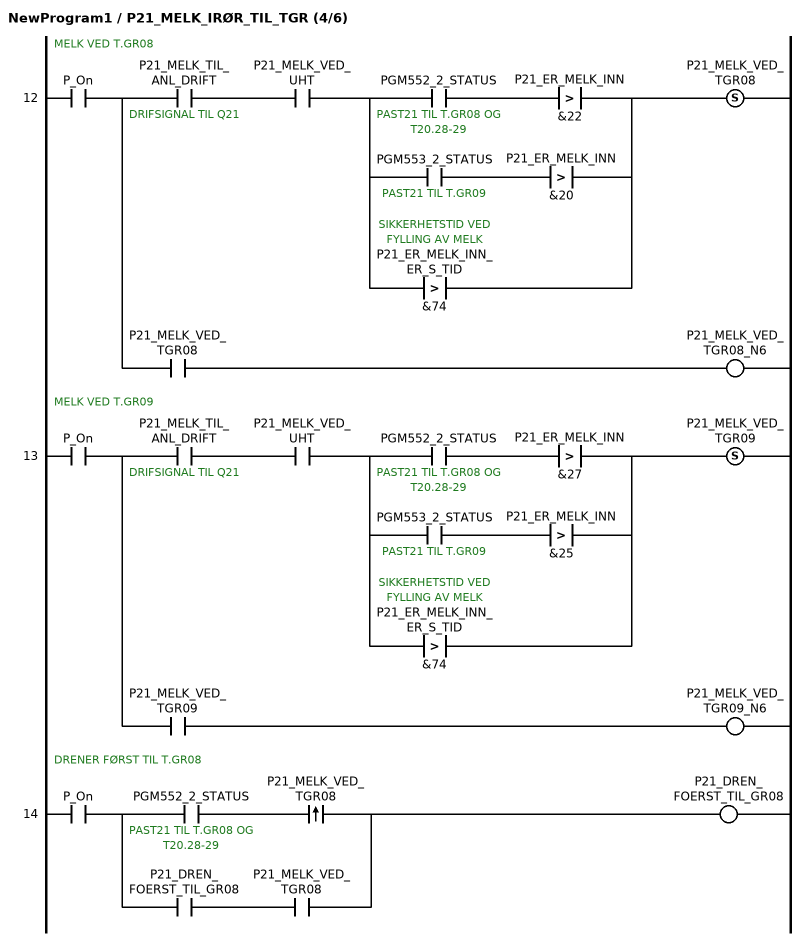
; rung 12: MELK VED T.GR08
LD P_On
OUT TR0
AND P21_MELK_TIL_ANL_DRIFT  ; DRIFSIGNAL TIL Q21
AND P21_MELK_VED_UHT
LD PGM552_2_STATUS  ; PAST21 TIL T.GR08 OG T20.28-29
AND>L(321) P21_ER_MELK_INN &22
LD PGM553_2_STATUS  ; PAST21 TIL T.GR09
AND>L(321) P21_ER_MELK_INN &20
ORLD
OR>(320) P21_ER_MELK_INN_ER_S_TID &74  ; SIKKERHETSTID VED FYLLING AV MELK
ANDLD
SET P21_MELK_VED_TGR08
LD TR0
AND P21_MELK_VED_TGR08
OUT P21_MELK_VED_TGR08_N6
; rung 13: MELK VED T.GR09
LD P_On
OUT TR0
AND P21_MELK_TIL_ANL_DRIFT  ; DRIFSIGNAL TIL Q21
AND P21_MELK_VED_UHT
LD PGM552_2_STATUS  ; PAST21 TIL T.GR08 OG T20.28-29
AND>L(321) P21_ER_MELK_INN &27
LD PGM553_2_STATUS  ; PAST21 TIL T.GR09
AND>L(321) P21_ER_MELK_INN &25
ORLD
OR>(320) P21_ER_MELK_INN_ER_S_TID &74  ; SIKKERHETSTID VED FYLLING AV MELK
ANDLD
SET P21_MELK_VED_TGR09
LD TR0
AND P21_MELK_VED_TGR09
OUT P21_MELK_VED_TGR09_N6
; rung 14: DRENER FØRST TIL T.GR08
LD P_On
LD PGM552_2_STATUS  ; PAST21 TIL T.GR08 OG T20.28-29
@AND P21_MELK_VED_TGR08
LD P21_DREN_FOERST_TIL_GR08
AND P21_MELK_VED_TGR08
ORLD
ANDLD
OUT P21_DREN_FOERST_TIL_GR08

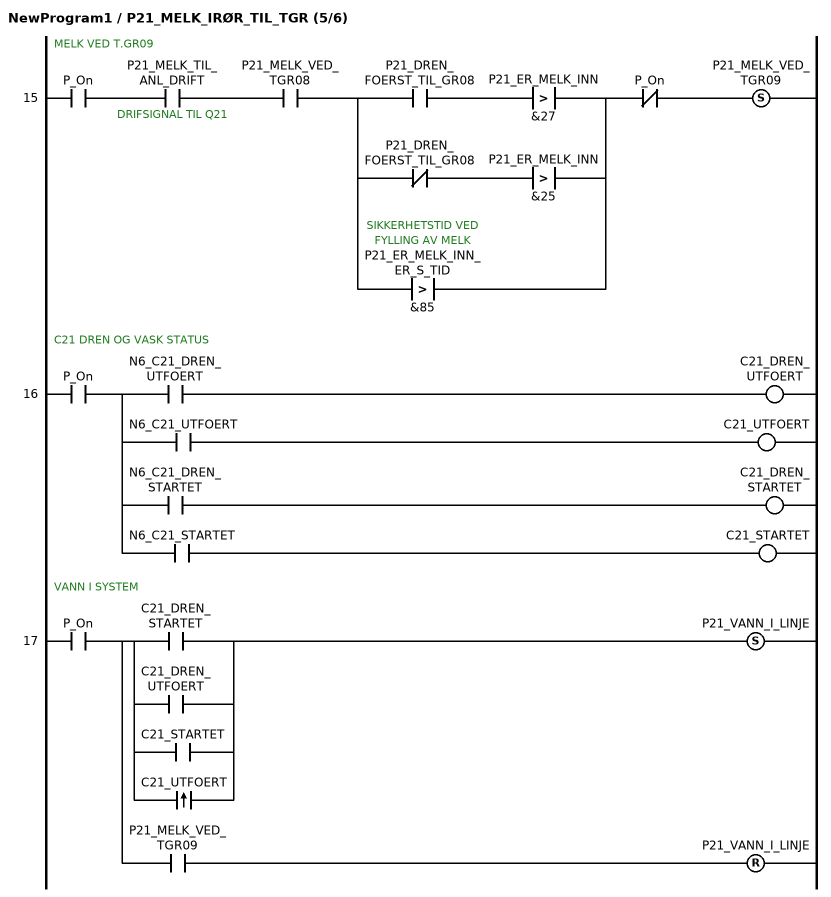
; rung 15: MELK VED T.GR09
LD P_On
AND P21_MELK_TIL_ANL_DRIFT  ; DRIFSIGNAL TIL Q21
AND P21_MELK_VED_TGR08
LD P21_DREN_FOERST_TIL_GR08
AND>L(321) P21_ER_MELK_INN &27
LDNOT P21_DREN_FOERST_TIL_GR08
AND>L(321) P21_ER_MELK_INN &25
ORLD
OR>(320) P21_ER_MELK_INN_ER_S_TID &85  ; SIKKERHETSTID VED FYLLING AV MELK
ANDLD
ANDNOT P_On
SET P21_MELK_VED_TGR09
; rung 16: C21 DREN OG VASK STATUS
LD P_On
OUT TR0
AND N6_C21_DREN_UTFOERT
OUT C21_DREN_UTFOERT
LD TR0
AND N6_C21_UTFOERT
OUT C21_UTFOERT
LD TR0
AND N6_C21_DREN_STARTET
OUT C21_DREN_STARTET
LD TR0
AND N6_C21_STARTET
OUT C21_STARTET
; rung 17: VANN I SYSTEM
LD P_On
OUT TR0
LD C21_DREN_STARTET
OR C21_DREN_UTFOERT
OR C21_STARTET
@OR C21_UTFOERT
ANDLD
SET P21_VANN_I_LINJE
LD TR0
AND P21_MELK_VED_TGR09
RSET P21_VANN_I_LINJE

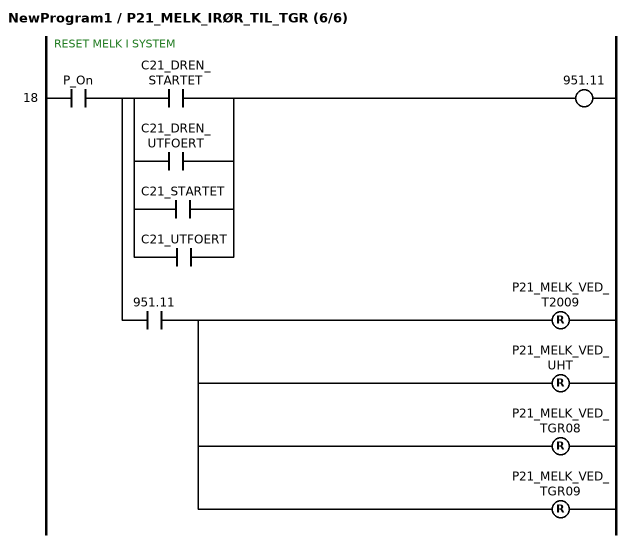
; rung 18: RESET MELK I SYSTEM
LD P_On
OUT TR0
LD C21_DREN_STARTET
OR C21_DREN_UTFOERT
OR C21_STARTET
OR C21_UTFOERT
ANDLD
OUT 951.11
LD TR0
AND 951.11
RSET P21_MELK_VED_T2009
RSET P21_MELK_VED_UHT
RSET P21_MELK_VED_TGR08
RSET P21_MELK_VED_TGR09

### Section HOMO21

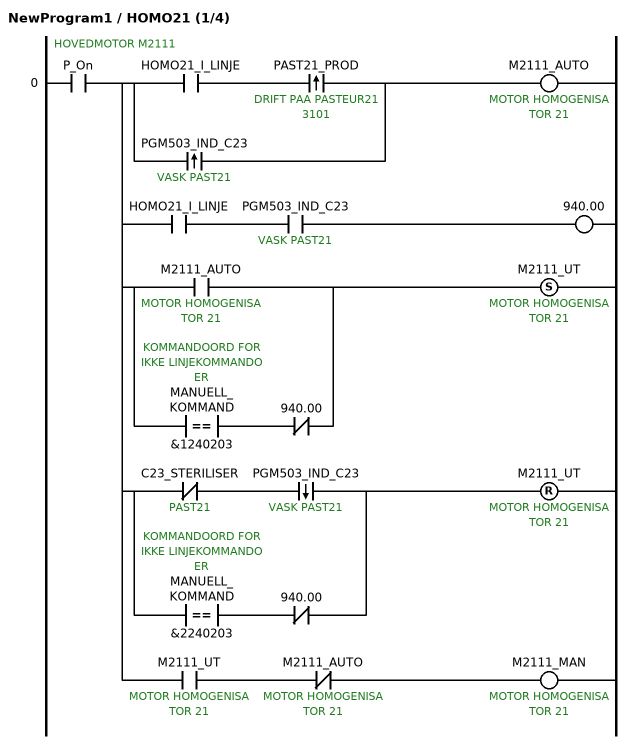
; rung 0: HOVEDMOTOR M2111
LD P_On
OUT TR0
LD HOMO21_I_LINJE
@AND PAST21_PROD  ; DRIFT PAA PASTEUR21 3101
@OR PGM503_IND_C23  ; VASK PAST21
ANDLD
OUT M2111_AUTO  ; MOTOR HOMOGENISATOR 21
LD TR0
AND HOMO21_I_LINJE
AND PGM503_IND_C23  ; VASK PAST21
OUT 940.00
LD TR0
LD M2111_AUTO  ; MOTOR HOMOGENISATOR 21
LD=L(301) MANUELL_KOMMAND &1240203  ; KOMMANDOORD FOR IKKE LINJEKOMMANDOER
ANDNOT 940.00
ORLD
ANDLD
SET M2111_UT  ; MOTOR HOMOGENISATOR 21
LD TR0
LDNOT C23_STERILISER  ; PAST21
%AND PGM503_IND_C23  ; VASK PAST21
LD=L(301) MANUELL_KOMMAND &2240203  ; KOMMANDOORD FOR IKKE LINJEKOMMANDOER
ANDNOT 940.00
ORLD
ANDLD
RSET M2111_UT  ; MOTOR HOMOGENISATOR 21
LD TR0
AND M2111_UT  ; MOTOR HOMOGENISATOR 21
ANDNOT M2111_AUTO  ; MOTOR HOMOGENISATOR 21
OUT M2111_MAN  ; MOTOR HOMOGENISATOR 21

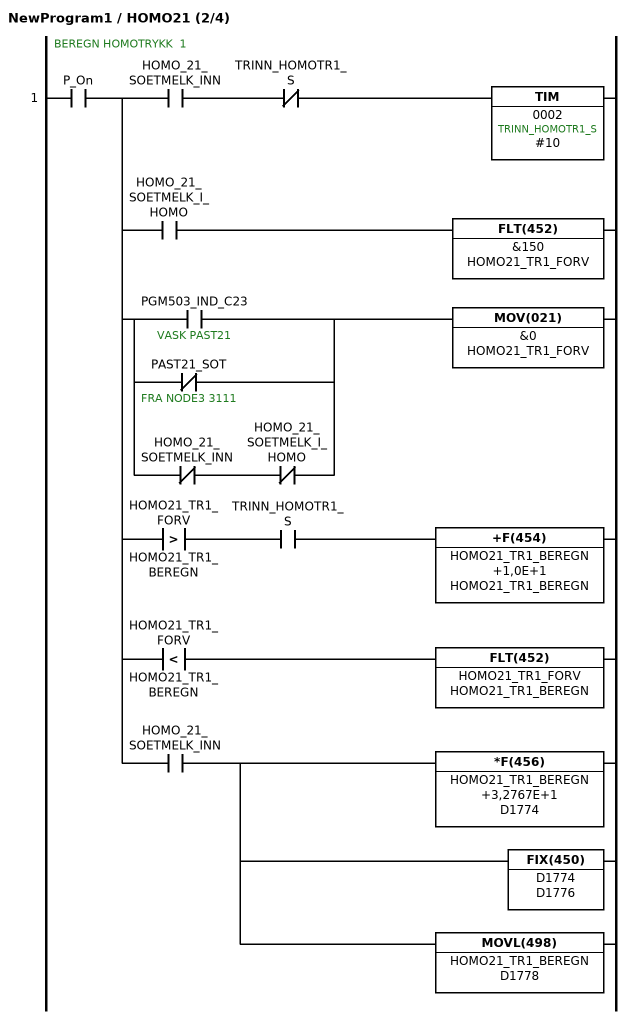
; rung 1: BEREGN HOMOTRYKK  1
LD P_On
OUT TR0
AND HOMO_21_SOETMELK_INN
ANDNOT TRINN_HOMOTR1_S
TIM 0002 #10  ; TRINN_HOMOTR1_S
LD TR0
AND HOMO_21_SOETMELK_I_HOMO
FLT(452) &150 HOMO21_TR1_FORV
LD TR0
LD PGM503_IND_C23  ; VASK PAST21
ORNOT PAST21_SOT  ; FRA NODE3 3111
LDNOT HOMO_21_SOETMELK_INN
ANDNOT HOMO_21_SOETMELK_I_HOMO
ORLD
ANDLD
MOV(021) &0 HOMO21_TR1_FORV
LD TR0
AND>F(333) HOMO21_TR1_FORV HOMO21_TR1_BEREGN
AND TRINN_HOMOTR1_S
+F(454) HOMO21_TR1_BEREGN +1,0E+1 HOMO21_TR1_BEREGN
LD TR0
AND<F(331) HOMO21_TR1_FORV HOMO21_TR1_BEREGN
FLT(452) HOMO21_TR1_FORV HOMO21_TR1_BEREGN
LD TR0
AND HOMO_21_SOETMELK_INN
*F(456) HOMO21_TR1_BEREGN +3,2767E+1 D1774
FIX(450) D1774 D1776
MOVL(498) HOMO21_TR1_BEREGN D1778

